{attribute addProperty BoxType "KL6211-0024"}
{attribute addProperty Id "Channel_1Channel_E2F3541B00"}
{attribute addProperty CRC "1878816392"}
{attribute addProperty SizeInBites "0"}
{attribute addProperty SizeInBytes "0"}
TYPE KL_6FFC7688 :
STRUCT
	{attribute addProperty Name "Channel_1"}
	Channel_1 : Channel_E2F3541B;
END_STRUCT
END_TYPE

(* stored: Version 1.2.0.0, ProductVersion 3.1.4024.9
   DUT KL_6FFC7688: Id {56961bc0-ed1b-4c83-a58e-90475054a859} *)
